Universal Robots PolyScope program: sprayRebate.urp

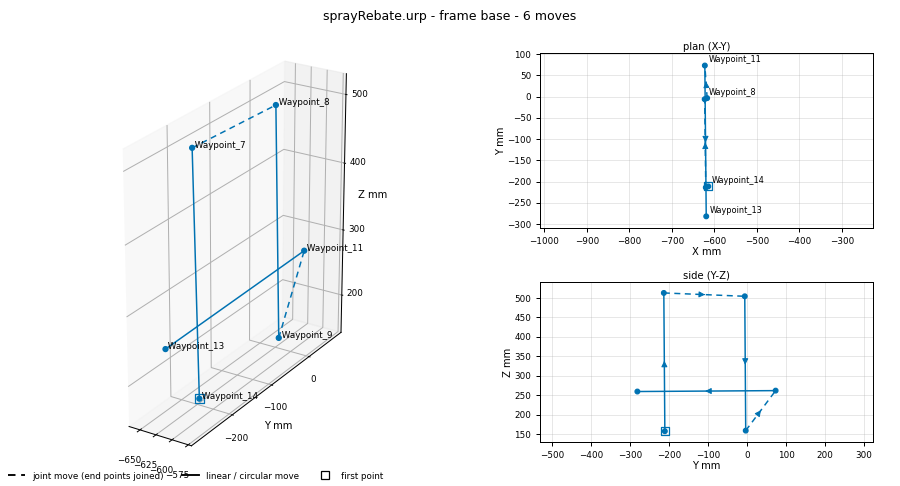
[picture p0: tool path of sprayRebate.urp in frame base, 6 of 6 moves have a stored position in this frame; points joined in program order, loops and branches not executed]
Program sprayRebate (installation=April22Cube directory=/programs/April2022Sand/subs createdIn=5.11.5.1010327 lastSavedIn=5.11.5.1010327 robotSerialNumber=20215500677)
Calibrated DH parameters: a=[0.000204, -0.239222, -0.391845, -0.000001, 0.000022, 0]; d=[0.162722, -355.808559, 353.37206, 2.570385, 0.099741, 0.099629]; alpha=[1.571124, 0.000988, 0.008295, 1.568963, -1.570303, 0]; deltaTheta=[0, -0.973091, 7.204745, 0.05153, 0, 0]
Robot Program (runOnlyOnce=false)
  Folder SprayRebate
    MoveJ speed 60 deg/s, acceleration 80 deg/s^2 (useActiveTCP=false) tcp=SprayTCP; feature=CubeFront
      Waypoint Waypoint_14: TCP in base x=-614.395 y=-211.304 z=158.056 mm, rx=0.8919 ry=-1.3989 rz=0.8972 rad; joints [3.832, -69.113, 116.159, -49.553, 73.09, -85.388] deg; TCP offset x=20.839 y=-27.14 z=105.994 mm, rx=0.1226 ry=1.1769 rz=2.8697 rad; feature pose in base x=-150.564 y=-110.257 z=792.369 mm, rx=-0.0207 ry=-0.0133 rz=3.0697 rad
      Set DigitalOutput pin=SprayerOn; digitalValue=1
    MoveL speed 100 mm/s, acceleration 1200 mm/s^2 (useActiveTCP=true) feature=CubeFront
      Waypoint Waypoint_7: TCP in base x=-620.397 y=-213.913 z=513.046 mm, rx=0.892 ry=-1.3988 rz=0.8971 rad; joints [4.169, -85.315, 79.236, 3.53, 73.033, -85.264] deg
      Set DigitalOutput pin=SprayerOn; digitalValue=0
      MoveDirectionNode (selectedDirection=ZPlus toolParams=0.2, 1.2)
        Until DISTANCE (allowActions=false deceleration=3 distanceNodeType=STOP) Distance=0.1; motionParameters(blendRadius=0)
    MoveJ speed 60 deg/s, acceleration 80 deg/s^2 (useActiveTCP=false) tcp=SprayTCP; feature=CubeFront
      Waypoint Waypoint_8: TCP in base x=-623.058 y=-6.085 z=504.453 mm, rx=-1.5379 ry=0.9456 rz=1.5188 rad; joints [-11.433, -87.799, 86.311, 5.702, 98.013, 93.92] deg
      Set DigitalOutput pin=SprayerOn; digitalValue=1
    MoveL speed 100 mm/s, acceleration 1200 mm/s^2 (useActiveTCP=false) tcp=SprayTCP; feature=CubeFront
      Waypoint Waypoint_9: TCP in base x=-617.186 y=-3.636 z=159.537 mm, rx=-1.538 ry=0.9455 rz=1.5188 rad; joints [-11.994, -68.384, 119.511, -46.936, 97.835, 93.758] deg
      Set DigitalOutput pin=SprayerOn; digitalValue=0
      MoveDirectionNode (selectedDirection=ZPlus toolParams=0.2, 1.2)
        Until DISTANCE (allowActions=false deceleration=3 distanceNodeType=STOP) Distance=0.1; motionParameters(blendRadius=0)
    MoveJ speed 60 deg/s, acceleration 80 deg/s^2 (useActiveTCP=false) tcp=SprayTCP; feature=CubeFront
      Waypoint Waypoint_11: TCP in base x=-622.643 y=73.149 z=262.251 mm, rx=2.0067 ry=-1.985 rz=-0.4223 rad; joints [-27.089, -68.36, 126.552, 146.432, -61.498, -7.368] deg; TCP offset x=20.839 y=-27.14 z=105.994 mm, rx=0.1226 ry=1.1769 rz=2.8697 rad
      Set DigitalOutput pin=SprayerOn; digitalValue=1
    MoveL speed 100 mm/s, acceleration 1200 mm/s^2 (useActiveTCP=false) tcp=SprayTCP; feature=CubeFront
      Waypoint Waypoint_13: TCP in base x=-619.354 y=-281.828 z=259.921 mm, rx=2.0066 ry=-1.9851 rz=-0.4224 rad; joints [19.517, -59.938, 112.11, 150.357, -104.552, 371.006] deg; TCP offset x=20.839 y=-27.14 z=105.994 mm, rx=0.1226 ry=1.1769 rz=2.8697 rad
      Set DigitalOutput pin=SprayerOn; digitalValue=0
      MoveDirectionNode (selectedDirection=ZPlus toolParams=0.2, 1.2)
        Until DISTANCE (allowActions=false deceleration=3 distanceNodeType=STOP) Distance=0.1; motionParameters(blendRadius=0)
